FUNCTION_BLOCK FB_PU_Schuetz_Output
VAR_INPUT
	Stellung			: BOOL;
END_VAR
VAR_OUTPUT
	OUT_Stellung	: BOOL;
END_VAR
VAR
END_VAR

OUT_Stellung := Stellung;

END_FUNCTION_BLOCK

(* stored: Version 1.1.0.1, ProductVersion 3.1.4024.9
   POU FB_PU_Schuetz_Output: Id {c1e26745-fd91-47ab-bf4b-0bb432bbd5ad}, SpecialFunc None *)
